//{attribute 'qualified_only'}
{attribute 'strict'}
TYPE eManual_State_Machine :
(
	Manual_Stop_State 	:= 0 ,
	Manual_Init_State 	:= 1 ,
	Manual_Ready_State 	:= 2 

);
END_TYPE

(* stored: Version 1.1.0.1, ProductVersion 3.1.4024.3
   EnumerationTextList eManual_State_Machine: Id {c3ea76fb-78b1-43a9-b690-c3de39a81793} *)
